FUNCTION_BLOCK MyControlClass
VAR
END_VAR

END_FUNCTION_BLOCK

(* stored: Version 1.1.0.1, ProductVersion 3.1.4024.12
   POU MyControlClass: Id {22f84247-0a53-41b5-853f-1172464fa996}, SpecialFunc None *)
